Fanuc KAREL source: kt00445.KL

-- PROVISIONAL review KL for V940-1; original PC SHA256 04fbf6754e95dacb7a20e9ad0ce9599727939a990615797669f07320e1af5b21
-- Incomplete behavior may be omitted. Consult companion uncertainty JSON. Do not deploy.
PROGRAM KT00445
%NOLOCKGROUP
VAR
  B1 : BOOLEAN
  B2 : BOOLEAN
  OUT : BOOLEAN
BEGIN
  -- V9_ZERO_TABLE_METADATA_HINT layout=0001; no indexed target words; source/name/runtime held
  -- UNRESOLVED_PC offsets 5-12; opcodes 9D,23
  -- UNRESOLVED_PC offsets 17-24; opcodes 9C,23
  -- UNRESOLVED_PC offsets 29-36; opcodes 9D,23
  -- UNRESOLVED_PC offsets 41-48; opcodes 9C,23
  -- UNRESOLVED_PC offsets 53-72; opcodes 21,21,5C,23
  -- UNRESOLVED_PC offsets 77-81; opcodes 7F
END KT00445
